PROGRAM FilterWheelControl
VAR_INPUT
	// move counter-clockwise
	left:	BOOL;
	// move clockwise
	right:	BOOL;
	// reset the axis(-error)
	reset:	BOOL;
	// enable the axis
	enable:	BOOL;
	// move to given psoition
	MoveAxis: BOOL;
	// calibrate the axis
	HomeAxis:	BOOL;
	// filter position
	filter_position: WORD;
END_VAR
VAR_OUTPUT
	error: 				BOOL;
	ErrorID:			UDINT;
	act_position:		LREAL;
END_VAR
VAR
	FilterWheelAxis:	FB_Axis2;
	position:			LREAL;
	FilterWheelEvent:	FB_EventLog;
END_VAR
VAR CONSTANT
	filters:	INT := 24;
END_VAR

(* This program controls the filter wheel. *)
enable := TelescopeControl.power OR PendantControl.FilterWheel_enable;

IF FilterWheelAxis.Calibrated THEN
	HomeAxis := FALSE;
	// limit filter_position to [0...filters-1]
	filter_position := filter_position MOD filters;
	position := 360.0 * INT_TO_LREAL(filter_position) / INT_TO_LREAL(filters);
ELSE
	position := 0.0;
	HomeAxis := TRUE;
END_IF

FilterWheelAxis(
	Enable := 			enable,
	Reset := 			reset,
	MoveAxis :=			MoveAxis,
	HomeAxis :=			HomeAxis,
	Position := 		position, 
	Enable_Positive :=  TRUE,
	Enable_Negative := 	TRUE,
	Jog_Forward :=		left,
	Jog_Backwards := 	right,
	bCalibrationCam :=	NOT GVL_FilterWheel.bCalibrationCam,
	isModuloAxis :=		TRUE,
	ActualPosition => 	act_position,
	Error => 			error,
	ErrorID => 			ErrorID,
	AxisRef :=			GVL_FilterWheel.FilterWheel_AxisRef);

IF FilterWheelAxis.MoveDone THEN
	MoveAxis := FALSE;
END_IF

IF FilterWheelAxis.HomeDone THEN
	HomeAxis := FALSE;
END_IF
	
IF FilterWheelAxis.ResetDone THEN
	reset := FALSE;
END_IF

FilterWheelEvent(	
	Trigger := 		Error, 
	Level := 		ADSLOG_MSGTYPE_ERROR,
	FormatString :=	'Filter Wheel Axis Error: %s',
	OnMessage := 	DWORD_TO_HEXSTR(ErrorID, 4, FALSE),
	OffMEssage := 	'OK',
	OffLevel := 	ADSLOG_MSGTYPE_HINT);

END_PROGRAM

(* stored: Version 1.1.0.1, ProductVersion 3.1.4024.4
   POU FilterWheelControl: Id {f0e4f375-0934-4386-a9fa-94537c34c7e1}, SpecialFunc None *)
